FUNCTION_BLOCK speedFbAdapter (* Retorno de velocidade: sinal normal (VTQREAL) ou valor bruto UINT16 com escala *)
  (* Standard: 61499-2 *)
  (* Version 1.0, 10/5/2026, Hidryco, Hidryco, Velocidade em INT para os sopradores Sulzer *)
  PACKAGE SE.Nereda;
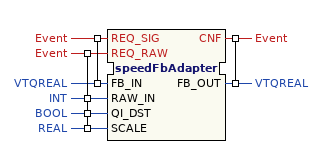
  EVENT_INPUT
    REQ_SIG WITH FB_IN;
    REQ_RAW WITH RAW_IN, QI_DST, SCALE;
  END_EVENT
  EVENT_OUTPUT
    CNF WITH FB_OUT;
  END_EVENT
  VAR_INPUT
    FB_IN : VTQREAL; (* Saida do aISignal fbSpeed *)
    RAW_IN : INT; (* Valor bruto do symlink fbSpeedINT *)
    QI_DST : BOOL; (* QO do SYMLINKMULTIVARDST (TRUE = conectado) *)
    SCALE : REAL; (* Fator: % = bruto / SCALE *)
  END_VAR
  VAR_OUTPUT
    FB_OUT : VTQREAL; (* Retorno de velocidade *)
  END_VAR
  VAR
    USE_RAW : BOOL;
    r : REAL;
  END_VAR
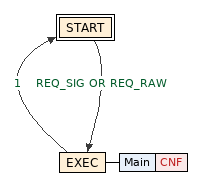
  EC_STATES
    START; (* Initial State *)
    EXEC : Main -> CNF;
  END_STATES
  EC_TRANSITIONS
    START TO EXEC := REQ_SIG OR REQ_RAW;
    EXEC TO START := 1;
  END_TRANSITIONS
  ALGORITHM Main IN ST:
(* Retorno de velocidade: usa o valor bruto INT do equipamento (fbSpeedINT) quando
   esse symlink esta conectado; senao repassa o rawPv/aISignal normal (fbSpeed.AIn).
   Valor bruto tratado como UINT16 e dividido por SCALE para voltar a %. *)
IF REQ_RAW AND QI_DST THEN
    USE_RAW := TRUE;
    r := INT_TO_REAL(RAW_IN);
    IF r < 0.0 THEN
        r := r + 65536.0;
    END_IF;
    IF SCALE > 0.0 THEN
        FB_OUT.value := r / SCALE;
    END_IF;
    FB_OUT.quality := 16#00000000;
ELSIF REQ_SIG AND NOT USE_RAW THEN
    FB_OUT := FB_IN;
END_IF;
  END_ALGORITHM
END_FUNCTION_BLOCK
